// TwinCAT 3 PLC project BottleSorter
// ProgramVersion: 3.1.4026.19
// libraries:
//   Tc2_Standard, * (Beckhoff Automation GmbH)
//   Tc2_System, * (Beckhoff Automation GmbH)
//   TcEventLogger, * (Beckhoff Automation Poland)
// project tree:
//   DUTs/ ST_Communication.TcDUT
//   GVLs/ GVL.TcGVL, GVL_Checks.TcGVL, GVL_Communication.TcGVL, GVL_ErrorHandling.TcGVL, GVL_IO.TcGVL, GVL_Recipe.TcGVL, GVL_StandAloneUnit.TcGVL, GVL_Unit.TcGVL, GVL_VIS.TcGVL
//   / PlcTask.TcTTO
//   POUs/ MAIN.TcPOU
// (motion and I/O tree: see PLC project programplc)
// real-time tasks:
//   TASK MainTask: cycle T#3ms, priority 20, ADS port 350
//   TASK SafetyTask: cycle T#10ms, priority 22, ADS port 351
//   TASK WeightTask: cycle T#2ms, priority 19, ADS port 354
//   TASK PlcTask: cycle T#10ms, priority 21, ADS port 355
//   TASK TaskToRefreshEAP: cycle T#1ms, priority 12, ADS port 301
// variable links:

CONFIGURATION BottleSorter
    RESOURCE PLC ON TwinCAT3
        TASK PlcTask(INTERVAL := T#10ms, PRIORITY := 21);
        PROGRAM MAIN WITH PlcTask : MAIN;
    END_RESOURCE
END_CONFIGURATION

// ---- DUTs/ST_Communication.TcDUT
TYPE ST_Communication :
STRUCT
	

	
	bEnable							: BOOL;	
	bCycleStart						: BOOL;
	bCycleStop						: BOOL;
	bCycleReset						: BOOL;
	bManualMode						: BOOL;
	bHoming							: BOOL;
	bHomingDone						: BOOL;	
	bConfectionEnding				: BOOL;
	tCycleTime						: TIME;
	iWatchdog						: INT;
	
	sRecipeName						: STRING(255);							
	sRecipeIndex					: STRING(255);

END_STRUCT
END_TYPE

// ---- GVLs/GVL.TcGVL
{attribute 'qualified_only'}
VAR_GLOBAL
	iRunningMode								: INT	:= 1;					// Pozniej zastanowic sie gdzie to zostawic
END_VAR

// ---- GVLs/GVL_Checks.TcGVL
{attribute 'qualified_only'}
VAR_GLOBAL PERSISTENT
	dCheckBounds					: DINT;			// Licznik przekroczen zakresu indexow, np. tablic
	dCheckDivDInt					: DINT;			// Licznik prob dzielenia Dint przez 0
	dCheckDivLInt					: DINT; 		// Licznik prob dzielenia LInt przez 0
	dCheckDivLReal					: DINT; 		// Licznik prob dzielenia LREAL przez 0
	dCheckDivReal					: DINT; 		// Licznik prob dzielenia REAL przez 0
	dCheckRangeSigned				: DINT;			// Licznik przekroczen liczby znakowej
	dCheckRangeUnsigned				: DINT; 		// Licznik przekroczen liczby bezznakowej
END_VAR

// ---- GVLs/GVL_Communication.TcGVL
VAR_GLOBAL
	stWrite				AT%MB0		: ST_Communication;			//Wysyłane zmienne do BottleUnboxer
	stRead				AT%I*		: ST_Communication;			//Odczytane zmienne z BottleUnboxer

	// Sygnały pomocnicze
	bEnable									: BOOL;
	bCycleStart								: BOOL;
	bCycleStop								: BOOL;
	bCycleReset								: BOOL;
	bManualMode								: BOOL;
	bHoming									: BOOL;	
	bHomingDone								: BOOL;
	bConfectionEnding						: BOOL;	
	bHomingDialog							: BOOL;
	bHomingCanceled							: BOOL;
	bChooseRecipe							: BOOL;
	bSafetyState							: BOOL;
	bReset									: BOOL;					// reset bledow z XTS          
	bRunLock								: BOOL;					//Blokada pracy   
	bSafetyReset							: BOOL;   
	bRecipeLoading							: BOOL;					//Wystawiane jak receptura jest ładowana                                           	
	bEmptingMode							: BOOL;
	bDoorClose								: BOOL;
END_VAR

// ---- GVLs/GVL_ErrorHandling.TcGVL
{attribute 'qualified_only'}
VAR_GLOBAL
	//Zmienne obslugi bledow
	bError										: BOOL;														// Zmienna ogolna wystapienia bledu                                                                         							
	udiErrorID									: UDINT;													// Kod bledu 	
	sErrorDescription1							: STRING(200);												// Opis bledu 1
	sErrorDescription2							: STRING(200);												// Opis bledu 2
	sStationInError								: STRING(200);												// Nazwa stacji w bledzie
                                                 
                                                                        	

	tonResettingTime							: TON;														// Licznik odliczacy czas wykonywania procedury resetu
	
	iStep										: INT;														// Krok proedury czytania bledow 	

END_VAR


VAR_GLOBAL CONSTANT
	iErrorStructuresNumber						: INT					:= 9;								// Liczba strukur bledow stacji  w tym strukura bledow globalnych
END_VAR

// ---- GVLs/GVL_IO.TcGVL
VAR_GLOBAL
	
(*Wejscia DI  BC1 EK1911*)

IbPowerSupplyOK 					AT %I*		:BOOL;		//	Napięcie zasilania OK
IbDCSupply1OK 						AT %I*		:BOOL;		//	Zasilacz 10G1 OK
IbFuse10F3							AT %I*		:BOOL;		//	Blok bezpiecznikowy 10F3 OK
IbFuse10F5							AT %I*		:BOOL;		//	Blok bezpiecznikowy 10F5 OK
IbDCSupply2OK 						AT %I*		:BOOL;		//	Zasilacz 10G2 OK
ibDCSupply5VDC_OK					AT %I*		: BOOL;		// Zasilanie 5VDC OK

(* DI1 EL1008*)

IbFuseDrivesOK						AT %I*		:BOOL;		//	Zabezpieczenie Servonapędu
IbFuseTransporter					AT %I*		:BOOL;		//	Zabezpieczenie transportera modulowego
IbEmergencyStop1Active				AT %I* 		:BOOL;		//	Aktywowany przycisk zatrzymania awaryjnego Estop poniżej szafy sterowniczej
IbEmergencyStop2Active				AT %I* 		:BOOL;		//	Aktywowany przycisk zatrzymania awaryjnego Estop przy zasypie zamkniec
IbEmergencyStop3Active				AT %I* 		:BOOL;		//	Aktywowany przycisk zatrzymania awaryjnego Estop przy zasypie zamkniec	


IbSafetyDoorOpen1					AT %I*		:BOOL;		//	Otwarte drzwi 1
IbSafetyDoorOpen2					AT %I*		:BOOL;		//	Otwarte drzwi 2
QbSafetyDoorOpen					AT %Q*		:BOOL;		//	Otwarcie drzwi

(*Wyjscia DQ*)
QbResetFuse10F3						AT %Q*		:BOOL;		// Reset bloku bezpiecznikowego 10F3
QbResetFuse10F5						AT %Q*		:BOOL;		// Reset bloku bezpiecznikowego 10F5

QbBackLight							AT %Q*		:BOOL;		// Załaczenie podświetlenia koła

// Obsluga pompy prozniowej
QbVacumPumpEnable				AT %Q*		: BOOL;		// Zalaczenie pompy prozniowej
IbFuseVacumPump					AT %I*		: BOOL;		//	Zabezpieczenie pompa prozniowa	
IbVacumPumpSensor				AT %I*		: BOOL;		//Czujnik cisnienia pompa prozniowa

//Obsługa zasilania w powietrze	
IbAirSupplyOK					AT %I*		: BOOL;		// Presostat powietrza
QbAirSupply						AT %Q*		: BOOL;		// Załączanie powietrza

//Błąd działania ProfiNet
IuiProfiNetError				AT %I*		: UINT;		// Błąd komunikacji ProfiNet - 0 to OK
IuiPnIoBoxStatePickMaster		AT %I*		: UINT;		// Status komunikacji profinet
IuiPnIoBoxStateRobotABB			AT %I*		: UINT;		// Status komunikacji profinet

//Wymiana danych z robotem
QbRobotPlace1					AT %Q*		: BOOL;		// Zezwol na położenie na stlot 1 (wystawić dopiero po start w PackMlu
QbRobotPlace2					AT %Q*		: BOOL;		// Zezwol na położenie na stlot 2
QbRobotPlace3					AT %Q*		: BOOL;		// Zezwol na położenie na stlot 3
QbRobotPlace4					AT %Q*		: BOOL;		// Zezwol na położenie na stlot 4

QbRobotPlaceDoneAck1			AT %Q*		: BOOL;		// Potwierdzenie butelka odłożona 1
QbRobotPlaceDoneAck2			AT %Q*		: BOOL;		// Potwierdzenie butelka odłożona 2
QbRobotPlaceDoneAck3			AT %Q*		: BOOL;		// Potwierdzenie butelka odłożona 3
QbRobotPlaceDoneAck4			AT %Q*		: BOOL;		// Potwierdzenie butelka odłożona 4

QbRobotStepMode					AT %Q*		: BOOL;		// Praca krokowa

QbRobotService					AT %Q*		: BOOL;		// Przejście robota w tryb serwisowy - potrzebne do ManualMovements
{warnin: DO usuniecia}
QbRobotServicePlace1			AT %Q*		: BOOL;		// Ruch robota do stlot 1 
QbRobotServicePlace2			AT %Q*		: BOOL;		// Ruch robota do stlot 2
QbRobotServicePlace3			AT %Q*		: BOOL;		// Ruch robota do stlot 3
QbRobotServicePlace4			AT %Q*		: BOOL;		// Ruch robota do stlot 4

QbRobotServiceVacumOn			AT %Q*		: BOOL;		// Załącz vacum
QbRobotServiceRejectOn			AT %Q*		: BOOL;		// Załącz odrzut
{warnin: DO usuniecia}
QbRobotServiceGripper			AT %Q*		: BOOL;		// Pozycja ramienia
{warnin: DO usuniecia}
IbRobotQueueFull1				AT %I*		: BOOL;		// Butelka wyjęta z kolejki wykrytych (nie wiem po co to nam)
IbRobotQueueFull2				AT %I*		: BOOL;		// Butelka wyjęta z kolejki wykrytych (nie wiem po co to nam)
IbRobotQueueFull3				AT %I*		: BOOL;		// Butelka wyjęta z kolejki wykrytych (nie wiem po co to nam)

IbRobotPlaceDone1				AT %I*		: BOOL;		// Butelka odłożona 1
IbRobotPlaceDone2				AT %I*		: BOOL;		// Butelka odłożona 2
IbRobotPlaceDone3				AT %I*		: BOOL;		// Butelka odłożona 3
IbRobotPlaceDone4				AT %I*		: BOOL;		// Butelka odłożona 4
{warnin: DO usuniecia}
IbRobotPosAvailable1			AT %I*		: BOOL;		// Potwierdzenie przyjęcia pozycji Place1
IbRobotPosAvailable2			AT %I*		: BOOL;		// Potwierdzenie przyjęcia pozycji Place2
IbRobotPosAvailable3			AT %I*		: BOOL;		// Potwierdzenie przyjęcia pozycji Place3

IbRobotVacumOn					AT %I*		: BOOL;		//Sygnał załaczenia Vacum
IbRobotVacumLevelOk				AT %I*		: BOOL;		//Sygnał z czujnika Vacum

IbRobotAutoOn					AT %I*		: BOOL;
IbRobotEmmergencyStop			AT %I*		: BOOL;
IbRobotExecutionError			AT %I*		: BOOL;
IbRobotMotionSupTrig			AT %I*		: BOOL;		// Kolizja
IbRobotMotorsOnState			AT %I*		: BOOL;
IbRobotRevCounterLost			AT %I*		: BOOL;		//Brak kalibracji
IbRobotTaskExecuting			AT %I*		: BOOL;		//Program się wykonuje
IbRobotWriteAcces				AT %I*		: BOOL;		//Załaczony dostęp zdalny
IbRobotSMBBatteryChargeLow		AT %I*		: BOOL;		//Alarm baterii


IdiRobotUnitModeCurrent			AT %I*		: DINT;	
IdiRobotStateCurrent			AT %I*		: DINT;	
IdiRobotRobotStatus0			AT %I*		: INT;
IdiRobotRobotStatus1			AT %I*		: INT;
IbRobotRobotIdle				AT %I*		: BOOL;
IbRobotRobotError				AT %I*		: BOOL;
IbRobotRobotPMRTConnected		AT %I*		: BOOL;
IbRobotRobotHeartBeat			AT %I*		: BOOL;
IudiRobotActiveOrder			AT %I*		: UDINT;	
IudiRobotErrorCode				AT %I*		: UDINT;	
IudiRobotCurrentRecipeID		AT %I*		: UDINT;	
IdiRobotBottelsCount			AT %I*		: DINT;
IuiRobotFieldbusType			AT %I*		: UINT := 2;

QdiRobotUnitMode				AT %Q*		: DINT;	
QdiRobotCntrlCmd				AT %Q*		: DINT;	
QdiRobotRobotCmd0				AT %Q*		: INT;
QdiRobotRobotCmd1				AT %Q*		: INT;
QbRobotUnitModeChangeRequest	AT %Q*		: BOOL;	
QbRobotCmdChangeRequest			AT %Q*		: BOOL;	
QbRobotRequest					AT %Q*		: BOOL;	
QbRobotResetError				AT %Q*		: BOOL;	
QudiRobotRequestOrder			AT %Q*		: UDINT;	
QudiRobotRequestRecipeID		AT %Q*		: UDINT;	

QbRobotGetFlowCount				AT %Q*		: BOOL;

QbEmptingDoorSolenoid			AT %Q*		: BOOL;

END_VAR

// ---- GVLs/GVL_Recipe.TcGVL
(*
Nazwa:			GVL_Recipe
Opis:			Zmienne recepturowe tylko do wizualizacji
Wersja:			v0.2
Data:			2024-02-20
Autor:			AS
Urzadzenia:		
Konfiguracja:	
Info:
Zmiany:
- 20240220 [DP] Poprawki przed nowa wizką
*)

{attribute 'qualified_only'}
VAR_GLOBAL
	(*Legenda dla wizki :
		[H] - Hidden, prawdopodobnie nie potrzebne
		[I] - Info, informacja,
		[L] - Later, do zrobienia później, być może do przerobienia
		Uprawienia:
		brak opisu - operator
		[m] - Meechanik i powyżej
		[t] - Technolog i powyżej
		[s] - Serwis i powyżek
		[a] - Admin			
	*)	

(******BottleSupplySorter********)	
(*******************************BottleSupplySorter Product Type**************************************************************************)	
	//Sorter butelek, typ produktu
	iBottleSorterProductTypeShow												: INT;					// 		Typ produktu
	uiBottleSorterIndexShow														: DINT;					// 		Index butelki 	
	                                                                   
(*******************************BottleSupplySorterHopperTransporter**************************************************************************)	
	//Sorter butelek, transporter zasobnika
	bBottleSorterHopperTransporterEnableShow									: BOOL;					//  	Aktywacja
	iBottleSorterHopperConveyorRunningSpeedSVShow								: INT	:= 5;			// 		Prędkość | [%] (1-100)
	iBottleSorterHopperConveyorEmptyingSpeedSVShow								: INT	:= 7;			// 		Prędkość, opróżnianie	| [%] (1-100)
	iBottleSorterDistanceToFindElementOnTransferConveyorLimitRunningSVShow		: INT	:= 610; 		// 		Odległość do butelek | [mm] (10-10_000)                                  		
	iBottleSorterDistanceToFindElementOnTransferConveyorLimitEmptyingSVShow		: INT	:= 500; 		// 		Odległość do butelek - opróżnianie | [mm] (10-10_000)                                       		

(*******************************BottleSupplySorterTransferTransporter**************************************************************************)
	//Sorter butelek, transporter transferowy	
	bBottleSorterTransferTransporterEnableShow									: BOOL;					// 		Aktywacja
	iBottleSorterTransferConveyorRunningSpeedSVShow								: INT	:= 5;			// 		Prędkość | [%] (1-100)	
	iBottleSorterTransferConveyorEmptyingSpeedSVShow							: INT	:= 7;			// 		Prędkość, opróżnianie | [%] (1-100)
	iBottleSorterDistanceToFindElementOnSupplyConveyorDownstairsLimitSVShow		: INT	:= 600;			// 		Odległość do butelek - stop zasypu | [mm] (10-10_000)
                                                                               
(*******************************BottleSupplySorterSupplyTransporter**************************************************************************)	
	//Sorter butelek, transporter zasypowy
	bBottleSorterSupplyTransporterEnableShow									: BOOL;					// [H] 	Aktywacja
	uiBottleSorterSupplyTransporterRunningSpeedSVShow							: UINT	:= 1_000;		// 		Prędkość | [obr/min] (10-10_000)	
	uiBottleSorterSupplyTransporterEmptingSpeedSVShow							: UINT	:= 1_000;		// 		Prędkość, opróżnianie | [obr/min] (10-10_000)                                                                   
	lrBottleSorterModuloMoveOffsetSVShow										: LREAL;				// 		Kat sprawdzania | [°] (1-360)	                                                                            
	//Logika zasypu - warunek pierwszy	                                                            
	iBottleSorterSensorsCountFirstConditionSVShow								: INT;					// 		Limit butelek
	iBottleSorterSupplyTimeFirstConditionSVShow									: INT;					// 		Czas zasypu | [ms] (10-10_000)                                                                                                    		
	//Logika zasypu - warunek drugi	 	                                                                                       		
	iBottleSorterSensorsCountSecondConditionMinSVShow							: INT;					// 		Limit butelek, min
	iBottleSorterSensorsCountSecondConditionMaxSVShow							: INT;					// 		Limit butelek, max
	iBottleSorterSupplyTimeSecondConditionSVShow								: INT;					// 		Czas zasypu | [ms] (10-10_000)                                                                                                  		
	//Logika zasypu - warunek trzeci 	                                                                                       		
	iBottleSorterSensorsCountThirdConditionSVShow								: INT;					// 		Limit butelek
	iBottleSorterSupplyTimeThirdConditionSVShow									: INT;					// 		Czas zasypu | [ms] (10-10_000)
	                                                                            	
(*******************************BottleSupplySorterWheel**************************************************************************)	
	//Sorter butelek, Stól
	bBottleSorterWeelEnableShow													: BOOL;					// [H]	Aktywacja
	lrBottleSorterWheelSpeedSVShow												: LREAL := 20;			// 		Prędkość | [obr/min] (5-100)	            
	lrBottleSorterWheelEmptyingSpeedSVShow										: LREAL := 30;			// 		Prędkość, opróżnianie | [obr/min] (5-100)	
		
(*******************************BottleSupplySorterBrush**************************************************************************)		
	//Sorter butelek, szczotka
	bBottleSorterBrushEnableShow												: BOOL;					//		Aktywacja
	lrBottleSorterBrushHeightPositionSVShow										: LREAL := 71;			// 		Wysokosc | [mm] (10-200)	
	iBottleSorterBrushRunningSpeedSVShow										: INT; 		 			// 		Prędkość | [%] (1-100)	            
	iBottleSorterBrushEmptyingSpeedSVShow										: INT; 		 			// 		Prędkość, opróżnianie | [%] (1-100)                                                              		         	
	
(*********************************BottleSupplyRobot*******************************************************************)

	//Sorter butelek, robot
	bBottleSorterRobotEnableShow												: BOOL;					// 		Aktywacja     
	nBottleSorterRobotRecipeId													: UDINT;				//		Nr receptury                                                                   
	//Czasy przyssania i oddmuchu                                                                                                                              
	lrBottleSorterRemainingTimeToSuctionShow             						: LREAL;				// 		Wyprzedzenie przyssania | [ms] (0-200)
	lrBottleSorterSuckerSuctionTimeShow											: LREAL;				// 		Czas przyssania	| [ms] (10-1000)
    lrBottleSorterRemainingTimeToRejectShow             						: LREAL;				// 		Wuprzedzenie oddmuchu | [ms] (0-200)
	lrBottleSorterEjectorPulseShow                                       		: LREAL;				// 		Czas oddmuchu	| [ms] (10-1000)			                                                                                                    		                                                                                                        		
	//Pkt. poboru i dokładania                                                                                 		                                                                                                          		
	lrBottleSorterZPickAboveTheBottleSVShow										: LREAL;				// 		Wysokość pobierania butelki
	lrBottleSorterZPickMoveSVShow												: LREAL;				// 		Odległość zjazdu w dół łapanie butelki 	                                                                                               	   		                                                                                     		
	lrBottleSorterSafetyHeightSVShow											: LREAL	:= 150;  		// 		Wysokość obracania chwytaka | [mm] (0-1000)

(*********************************BottleReciever*******************************************************************)

	//Sorter butelek, robot
	bBottleSorterRecieverEnableShow												: BOOL;					// 		Aktywacja   
	bBottleSorterRecieverSlot1EnableShow										: BOOL;					// 		Aktywacja  
	bBottleSorterRecieverSlot2EnableShow										: BOOL;					// 		Aktywacja  
	bBottleSorterRecieverSlot3EnableShow										: BOOL;					// 		Aktywacja  
	lrBottleSorterRecieverHeightPositionSVShow									: LREAL;				// 		Wysokosc | [mm] (10-200)
                                                                   
	lrBottleSorterRecieverSlotPositionSVShow									: LREAL;				
	lrBottleSorterRecieverMiddlePositionSVShow									: LREAL;				
	lrBottleSorterRecieverPuckPositionSVShow									: LREAL;				

END_VAR

// ---- GVLs/GVL_StandAloneUnit.TcGVL
{attribute 'qualified_only'}
VAR_GLOBAL
	bStandAlone									: BOOL;		// Without superior system
	bNoPackML									: BOOL;		// Without PackML
	bGhostMode									: BOOL; 	// Without product, demo mode
	bStartCycle									: BOOL;
	bStopCycle									: BOOL;
	bServiceMode								: BOOL;
	bHoming										: BOOL;
	bReset										: BOOL;
	bChooseRecipe								: BOOL;
	bProductionEnding							: BOOL;
	bDoorOpen									: BOOL;
	
END_VAR

// ---- GVLs/GVL_Unit.TcGVL
{attribute 'qualified_only'}
VAR_GLOBAL
																							
END_VAR

// ---- GVLs/GVL_VIS.TcGVL
(*
Nazwa:			GVL_VIS
Opis:			Zmienne dla wizualizacji
Wersja:			v0.2
Data:			2024-02-20
Autor:			AS
Urzadzenia:		
Konfiguracja:	
Info:
Zmiany:
- 20240220 [DP] Poprawki przed nowa wizką
*)

{attribute 'qualified_only'}
VAR_GLOBAL	
	
	(*Legenda dla wizki :
		[H] - Hidden, prawdopodobnie nie potrzebne
		[I] - Info, informacja,
		[L] - Later, do zrobienia później, być może do przerobienia
	Uprawienia:
		brak opisu - operator
		[m] - Meechanik i powyżej
		[t] - Technolog i powyżej
		[s] - Serwis i powyżek
		[a] - Admin			
	*)

(*******************************BottleSupplySorterHopperTransporters**************************************************************************)	
	//Sorter butelek, transporter zasobnika
	iBottleSorterHopperTransporterState						: INT;			// Stan
	sBottleSorterHopperTransporterState						: STRING;		// Stan
	bBottleSorterHopperTransporterHoming					: BOOL;			// Bazowanie					// Przycisk bistabilny
	bBottleSorterManualHopperConveyorForward				: BOOL;	  		// Do przodu					// Przycisk bistabilny
	iBottleSorterManualHopperConveyorSpeed					: INT;	  		// Prędkość | [%] (1-100)		// Pole do wpisywania wartosci
	iBottleSorterHopperConveyorSpeedCV						: INT;	  		// Predkosc aktualna | [%]		// Pole do wyświetlania wartości

	iDistanceToFindElementOnTransferConveyor				: INT;
	
(*******************************BottleSupplySorterTransferTransporter**************************************************************************)		
	//Sorter butelek, transporter transferowy	
	iBottleSorterTransferTransporterState					: INT;			// Stan
	sBottleSorterTransferTransporterState					: STRING;		// Stan
	bBottleSorterTransferTransporterHoming					: BOOL;			// Bazowanie					// Przycisk bistabilny
	bBottleSorterManualTransferConveyorForward				: BOOL;	  		// Do przodu					// Przycisk bistabilny
	bBottleSorterManualTransferConveyorBackward				: BOOL;	  		// Do tyłu						// Przycisk bistabilny	
	iBottleSorterManualTransferConveyorSpeed				: INT;	  		// Prędkość | [%] (1-100)		// Pole do wpisywania wartosci
	iBottleSorterTransferConveyorSpeedCV					: INT;	  		// Predkosc aktualna | [%]		// Pole do wyświetlania wartości
	
	iDistanceToFindElementOnSupplyConveyorDownstairs		: INT;
	
(*******************************BottleSupplySorterSupplyTransporter**************************************************************************)	
	//Sorter butelek, transporter zasypowy
	iBottleSorterSupplyTransporterState						: INT;			// Stan
	sBottleSorterSupplyTransporterState						: STRING;		// Stan
	bBottleSorterSupplyTransporterHoming					: BOOL;			// Bazowania							// Przycisk bistabilny
	bBottleSorterManualSupplyTransporterForward				: BOOL;	  		// Do przodu							// Przycisk monostabilny
	uiBottleSorterManualSupplyConveyorSpeed					: UINT;	  		// Prędkość | [obr/min] (10-10_000)		// Pole do wpisywania wartosci
	iBottleSorterSupplyConveyorSpeedCV						: INT;	  		// Predkosc aktualna | [obr/min]		// Pole do wyświetlania wartości
	
(*******************************BottleSupplySorterBrush**************************************************************************)	
	//Sorter butelek, szczotka
	iBottleSorterBrushState									: INT;			// Stan
	sBottleSorterBrushState									: STRING;       // Stan
	bBottleSorterBrushHoming								: BOOL;			// Bazowanie							// Przycisk bistabilny
	lrBottleSorterBrushHeightCV								: LREAL;  		// Aktualna wysokosc | [mm]				// Pole do wyświetlania wartości
	iBottleSorterBrushSpeedCV								: INT;	  		// Aktualna predkość | [%]				// Pole do wyświetlania wartości
    bBottleSorterBrushHeightSet         					: BOOL;   		// Ustaw 								// Przycisk monostabilny
	bBottleSorterManualBrushLiftUp							: BOOL;	  		// Do góry								// Przycisk monostabilny
	bBottleSorterManualBrushLiftDown						: BOOL;	  		// Do dołu								// Przycisk monostabilny
	bBottleSorterManualBrushDriveForward					: BOOL;	  		// Do przodu							// Przycisk bistabilny
	bBottleSorterManualBrushDriveBackward					: BOOL;	  		// Do tyłu								// Przycisk bistabilny
	iBottleSorterManualBrushSpeedSV							: INT;  		// Prędkość |[%] (1-100)				// Pole do wpisywania wartosci
	
(*******************************BottleSupplySorterWheel**************************************************************************)	
	//Sorter butelek, stół
	iBottleSorterWheelState									: INT;			// Stan
	sBottleSorterWheelState									: STRING;       // Stan
	bBottleSorterWheelHoming								: BOOL;			// Bazowanie							// Przycisk bistabilny
    bBottleSorterManualWheelRight    						: BOOL;   		// W prawo								// Przycisk monostabilny
    bBottleSorterManualWheelLeft     						: BOOL;   		// W lewo 								// Przycisk monostabilny
	bBottleSorterManualWheelFixedAngleMovement				: BOOL;			// Ustaw								// Przycisk monostabilny
	lrBottleSorterWheelSpeedCV								: LREAL;		// Aktualna predkość | [obr/min]		// Pole do wyświetlania wartości
	lrBottleSorterManualWehhelFIxedAngle					: LREAL := 110;	// Kąt obrotu | [°] (1-360)				// Pole do wpisywania wartosci
	lrBottleSorterManualWheelSpeed							: LREAL	:= 10;	// Prędkośc | [obr/min] (1-1000)		// Pole do wpisywania wartosci
	bBottleSorterManualWheelBarier  						: BOOL;   		// Otwórz/Zamknij						// Przycisk bistabilny	
	
	
(*********************************BottleSupplyRobot*******************************************************************)
	//Sorter butelek, robot
	iBottleSorterRobotState									: INT;			// Stan																
	sBottleSorterRobotState									: STRING;       // Stan
	bBottleSorterRobotHoming								: BOOL;			// Bazowanie				// Przycisk bistabilny	
	diBottleSorterRobotSpeed								: DINT; 		// Prędkość | [%] (1-100)	// Pole do wpisywania wartosci
	bBottleSorterRobotManualPlace1							: BOOL;			// Ruch robota do stlot 1
	bBottleSorterRobotManualPlace2							: BOOL;			// Ruch robota do stlot 2
	bBottleSorterRobotManualPlace3							: BOOL;			// Ruch robota do stlot 3
	bBottleSorterRobotManualVacumOn							: BOOL;			// Załącz vacum				// Przycisk bistabilny
	bBottleSorterRobotManualRejectOn						: BOOL;			// Załącz odrzut			// Przycisk bistabilny
	bBottleSorterRobotManualGripper							: BOOL;			// Pozycja ramienia			// Przycisk bistabilny

	bBottleSorterRobotActualRecipeID						: UDINT;		// Nr aktualnej receptury na robocie
	
(*********************************BottleReciever*******************************************************************)
	//Sorter butelek, robot
	iBottleSorterRecieverState									: UINT;			// Stan																
	sBottleSorterRecieverState									: STRING;       // Stan
	bBottleSorterRecieverHoming									: BOOL;			// Bazowanie				// Przycisk bistabilny		
	lrBottleSorterRecieverHeightPositionCV						: LREAL;		// Wysokosc | [mm] (10-200)
	bBottleSorterRecieverHeightSet         						: BOOL;   		// Ustaw 						// Przycisk monostabilny	
	bBottleSorterRecieverManualCatcherUp						: BOOL;			// Podnieś chwytaki butelek
	bBottleSorterRecieverManualCatcherDown						: BOOL;			// Opuść chwytaki butelek
	bBottleSorterRecieverManualCatcher1Open						: BOOL;			// Otwórz chwytak stały 1
	bBottleSorterRecieverManualCatcher2Open						: BOOL;			// Otwórz chwytak stały 2
	bBottleSorterRecieverManualCatcher3Open						: BOOL;			// Otwórz chwytak stały 3
	bBottleSorterRecieverManualCatcher1Close					: BOOL;			// Zamknij chwytak stały 1
	bBottleSorterRecieverManualCatcher2Close					: BOOL;			// Zamknij chwytak stały 2
	bBottleSorterRecieverManualCatcher3Close					: BOOL;			// Zamknij chwytak stały 3
	bBottleSorterRecieverManualGripper1Open						: BOOL;			// Otwórz chwytak ruchomy 1
	bBottleSorterRecieverManualGripper2Open						: BOOL;			// Otwórz chwytak ruchomy 2
	bBottleSorterRecieverManualGripper3Open						: BOOL;			// Otwórz chwytak ruchomy 3
	bBottleSorterRecieverManualGripper1Close					: BOOL;			// Zamknij chwytak ruchomy 1
	bBottleSorterRecieverManualGripper2Close					: BOOL;			// Zamknij chwytak ruchomy 2
	bBottleSorterRecieverManualGripper3Close					: BOOL;			// Zamknij chwytak ruchomy 3
	bBottleSorterRecieverManualVerticalUp						: BOOL;			// Podnieś chwytaki ruchome butelek
	bBottleSorterRecieverManualVerticalDown						: BOOL;			// Opuść chwytaki ruchome butelek
	bBottleSorterRecieverManualHotizontalIn						: BOOL;			// Przesuń chwytaki ruchome butelek
	bBottleSorterRecieverManualHotizontalOut					: BOOL;			// Przesuń chwytaki ruchome butelek
	bBottleSorterRecieverManualFormatCatched					: BOOL;			// Docisk formatek zamknięty
	bBottleSorterRecieverManualFormatRelised					: BOOL;			// Docisk formatek otwarty
	bBottleSorterRecieverManualFormatStoperOut					: BOOL;			// Szlaban formatek otwarty
	bBottleSorterRecieverManualFormatStoperIn					: BOOL;			// Szlaban formatek zamknięty
	bBottleSorterRecieverManualJisangUp							: BOOL;			// 
	bBottleSorterRecieverManualJisangDown						: BOOL;			// 
	
	bBottleSorterRecieverManualBottleHammerOn					: BOOL;			// 
	bBottleSorterRecieverManualSlotVacumOn						: BOOL;			// 
	bBottleSorterRecieverManualHotizontalMiddle					: BOOL;			// 
	bBottleSorterRecieverManualGrippersClose					: BOOL;			// 
	
	
	lrBottleSorterRecieverManualHeightPositionSV				: LREAL;		// 		Wysokosc | [mm] (10-200)
	fbAlarms 											:FB_Events;	
	//Poziomy zasypu
	bfewbottles													: BOOL;				
	bmorebottles                                                : BOOL;
	bmostbottles                                                : BOOL;
END_VAR

// ---- POUs/MAIN.TcPOU
PROGRAM MAIN
VAR
END_VAR

gvl.iRunningMode;
gvl_checks.dCheckBounds;
gvl_communication.bChooseRecipe;
gvl_errorHandling.bError;
gvl_io.IbAirSupplyOK;
gvl_recipe.bBottleSorterBrushEnableShow;
gvl_standaloneunit.bChooseRecipe;
gvl_vis.bBottleSorterBrushHeightSet;

END_PROGRAM
